PROGRAM MAIN
VAR
END_VAR

END_PROGRAM

(* stored: Version 1.1.0.1
   POU MAIN: Id {2cd28470-6329-4078-8e6a-d75c8e1492ad} *)
